// TIA Portal project "Soru2" (V15)

(* hardware
DEVICE "S7-1200 station_1"  S7-1200 Station
   slot 0: "Rack_0"  S7-1200 Rack  Rack  V1.0
   slot 1: "PLC_1"  CPU 1214C DC/DC/DC  6ES7 214-1AG40-0XB0  V4.2
*)

// ===== PLC "PLC_1"  CPU 1214C DC/DC/DC =====

VAR_GLOBAL   // PLC tag table "Default tag table"
   "GeceModu değil mi" AT %I0.0 : Bool;
   "Oto icin yeşil" AT %Q0.0 : Bool;
   "Oto icin sari" AT %Q0.1 : Bool;
   "Oto için kırmızı" AT %Q0.2 : Bool;
   "Yaya için yeşil" AT %Q0.3 : Bool;
   "Yaya için kımızı" AT %Q0.4 : Bool;
   "Pause Tuşu" AT %I0.1 : Bool;
END_VAR

// folder: System blocks/Program resources

DATA_BLOCK "OTO_VE_YAYA_yesil_kirimizi_H"   // DB2
{ S7_Optimized_Access := 'TRUE' }
AUTHOR : Simatic
FAMILY : IEC
NAME : IEC_TMR
VERSION : 1.0
// stored: InstanceOfName IEC_TIMER
"IEC_TIMER"
BEGIN
END_DATA_BLOCK

DATA_BLOCK "OTO_VE_YAYA_yesil_kirimizi_L"   // DB3
{ S7_Optimized_Access := 'TRUE' }
AUTHOR : Simatic
FAMILY : IEC
NAME : IEC_TMR
VERSION : 1.0
// stored: InstanceOfName IEC_TIMER
"IEC_TIMER"
BEGIN
END_DATA_BLOCK

DATA_BLOCK "Gece_mod_H"   // DB8
{ S7_Optimized_Access := 'TRUE' }
AUTHOR : Simatic
FAMILY : IEC
NAME : IEC_TMR
VERSION : 1.0
// stored: InstanceOfName IEC_TIMER
"IEC_TIMER"
BEGIN
END_DATA_BLOCK

DATA_BLOCK "Gece_mod_L"   // DB9
{ S7_Optimized_Access := 'TRUE' }
AUTHOR : Simatic
FAMILY : IEC
NAME : IEC_TMR
VERSION : 1.0
// stored: InstanceOfName IEC_TIMER
"IEC_TIMER"
BEGIN
END_DATA_BLOCK

DATA_BLOCK "OTO_sari_Ld"   // DB10
{ S7_Optimized_Access := 'TRUE' }
AUTHOR : Simatic
FAMILY : IEC
NAME : IEC_TMR
VERSION : 1.0
// stored: InstanceOfName IEC_TIMER
"IEC_TIMER"
BEGIN
END_DATA_BLOCK

DATA_BLOCK "OTO_sari_Hd"   // DB11
{ S7_Optimized_Access := 'TRUE' }
AUTHOR : Simatic
FAMILY : IEC
NAME : IEC_TMR
VERSION : 1.0
// stored: InstanceOfName IEC_TIMER
"IEC_TIMER"
BEGIN
END_DATA_BLOCK

// folder: (top level)

ORGANIZATION_BLOCK "Main"   // OB1, LAD, ProgramCycle
TITLE = "Main Program Sweep (Cycle)"
{ S7_Optimized_Access := 'TRUE' }
VERSION : 0.1
   VAR_INPUT
      Initial_Call : Bool;   // Initial call of this OB
      Remanence : Bool;   // =True, if remanent data are available
   END_VAR
BEGIN

REGION Network 1: Otolar için kırmızı ve yayalar için yeşil Zaman döngüsü
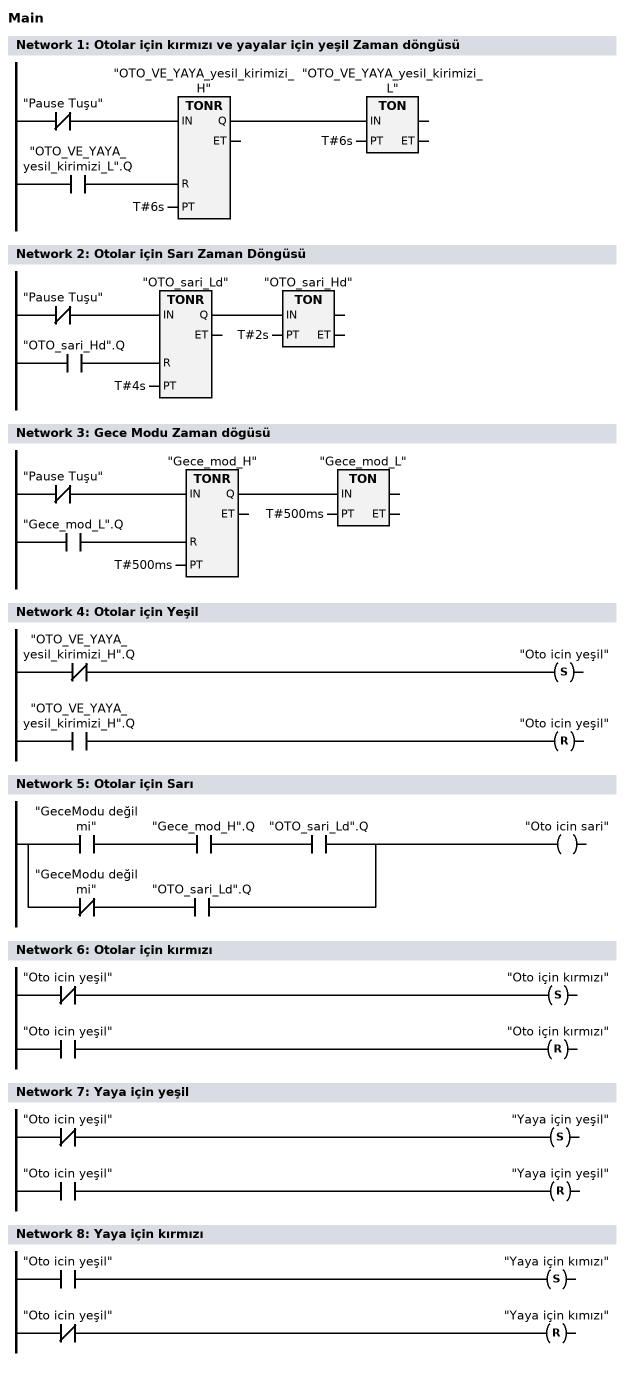
   "OTO_VE_YAYA_yesil_kirimizi_H".TONR(IN := NOT "Pause Tuşu",
                           R := "OTO_VE_YAYA_yesil_kirimizi_L".Q,
                           PT := T#6s);
   "OTO_VE_YAYA_yesil_kirimizi_L".TON(IN := "OTO_VE_YAYA_yesil_kirimizi_H".Q, PT := T#6s);
END_REGION

REGION Network 2: Otolar için Sarı Zaman Döngüsü
   "OTO_sari_Ld".TONR(IN := NOT "Pause Tuşu", R := "OTO_sari_Hd".Q, PT := T#4s);
   "OTO_sari_Hd".TON(IN := "OTO_sari_Ld".Q, PT := T#2s);
END_REGION

REGION Network 3: Gece Modu Zaman dögüsü
   "Gece_mod_H".TONR(IN := NOT "Pause Tuşu", R := "Gece_mod_L".Q, PT := T#500ms);
   "Gece_mod_L".TON(IN := "Gece_mod_H".Q, PT := T#500ms);
END_REGION

REGION Network 4: Otolar için Yeşil
   RUNG wire#powerrail
      I_Contact( "OTO_VE_YAYA_yesil_kirimizi_H".Q )
      S_Coil( "Oto icin yeşil" )
   END_RUNG
   RUNG wire#powerrail
      Contact( "OTO_VE_YAYA_yesil_kirimizi_H".Q )
      R_Coil( "Oto icin yeşil" )
   END_RUNG
   // the same network as SCL:
   IF NOT "OTO_VE_YAYA_yesil_kirimizi_H".Q THEN "Oto icin yeşil" := TRUE; END_IF;
   IF "OTO_VE_YAYA_yesil_kirimizi_H".Q THEN "Oto icin yeşil" := FALSE; END_IF;
END_REGION

REGION Network 5: Otolar için Sarı
   RUNG wire#powerrail
      Contact( "GeceModu değil mi" )
      Contact( "Gece_mod_H".Q )
      Contact( "OTO_sari_Ld".Q )
      wire#w1
      Coil( "Oto icin sari" )
   END_RUNG
   RUNG wire#powerrail
      I_Contact( "GeceModu değil mi" )
      Contact( "OTO_sari_Ld".Q )
   END_RUNG wire#w1
   // the same network as SCL:
   "Oto icin sari" := ("GeceModu değil mi" AND "Gece_mod_H".Q AND "OTO_sari_Ld".Q) OR (NOT "GeceModu değil mi" AND "OTO_sari_Ld".Q);
END_REGION

REGION Network 6: Otolar için kırmızı
   RUNG wire#powerrail
      I_Contact( "Oto icin yeşil" )
      S_Coil( "Oto için kırmızı" )
   END_RUNG
   RUNG wire#powerrail
      Contact( "Oto icin yeşil" )
      R_Coil( "Oto için kırmızı" )
   END_RUNG
   // the same network as SCL:
   IF NOT "Oto icin yeşil" THEN "Oto için kırmızı" := TRUE; END_IF;
   IF "Oto icin yeşil" THEN "Oto için kırmızı" := FALSE; END_IF;
END_REGION

REGION Network 7: Yaya için yeşil
   RUNG wire#powerrail
      I_Contact( "Oto icin yeşil" )
      S_Coil( "Yaya için yeşil" )
   END_RUNG
   RUNG wire#powerrail
      Contact( "Oto icin yeşil" )
      R_Coil( "Yaya için yeşil" )
   END_RUNG
   // the same network as SCL:
   IF NOT "Oto icin yeşil" THEN "Yaya için yeşil" := TRUE; END_IF;
   IF "Oto icin yeşil" THEN "Yaya için yeşil" := FALSE; END_IF;
END_REGION

REGION Network 8: Yaya için kırmızı
   RUNG wire#powerrail
      Contact( "Oto icin yeşil" )
      S_Coil( "Yaya için kımızı" )
   END_RUNG
   RUNG wire#powerrail
      I_Contact( "Oto icin yeşil" )
      R_Coil( "Yaya için kımızı" )
   END_RUNG
   // the same network as SCL:
   IF "Oto icin yeşil" THEN "Yaya için kımızı" := TRUE; END_IF;
   IF NOT "Oto icin yeşil" THEN "Yaya için kımızı" := FALSE; END_IF;
END_REGION
END_ORGANIZATION_BLOCK